# EPICS StreamDevice protocol: pfeiffer/tpg361/device_config/pfeiffertpg361.proto
Terminator = CR LF;

p_stat_get{
	out "PR1";
	in 0x06;
	out 0x05;
	in "%1d,%*e";
}

p_get_raw{
	#out "PR1";
	#in 0x06;
	#out 0x05;
	in "%*1d,%e";
}
